Staubli VAL3: onRightEvent.pgx

program onRightEvent()
  local num l_nDefault
  local num l_nSize
begin
  l_nSize=3
  // step -1
  call processList:getDefaultType(l_nDefault)
  l_nDefault=(l_nDefault+1)%(l_nSize)
  call processList:setDefaultType(l_nDefault)
  use:bUseRefresh=true
end
